// TIA Portal V18 export
FUNCTION_BLOCK "Block_1"   // FB8, SCL
{ S7_Optimized_Access := 'TRUE' }
// stored: AutoNumber false, MemoryReserve 1000, SetENOAutomatically false
BEGIN
END_FUNCTION_BLOCK
